TYPE M2MultiplexerStatuses :
STRUCT
	///Is the selected drive healthy?
	healthStatus: HealthStatus;
	///Is the selected drive busy?
	busyStatus: BusyStatus;
END_STRUCT
END_TYPE

(* stored: Version 1.1.0.1, ProductVersion 3.1.4019.2
   DUT M2MultiplexerStatuses: Id {e16cde86-bd27-4519-8bb7-ed955eeea6b2} *)
